TYPE Ed12dssShutterConfig EXTENDS DeviceConfiguration :
STRUCT	
END_STRUCT
END_TYPE

(* stored: Version 1.1.0.1, ProductVersion 3.1.4024.4
   DUT Ed12dssShutterConfig: Id {89a7dbef-e89c-4dda-a2b3-fa0778a27af4} *)
